Fanuc KAREL source: kb00029.KL

-- PROVISIONAL review KL for V770-1; original PC SHA256 8f31ae490222605812ec860d8ad9381e16546bc304840df08ca040dcb082aeb5
-- Incomplete behavior may be omitted. Consult companion uncertainty JSON. Do not deploy.
PROGRAM KB00029
%NOLOCKGROUP
BEGIN
  -- UNRESOLVED_PC offsets 5-12; opcodes 9D,23
  -- UNRESOLVED_PC offsets 17-26; opcodes 3F,75
  -- UNRESOLVED_PC offsets 31-38; opcodes 9D,23
  -- UNRESOLVED_PC offsets 43-67; opcodes 27,22,22,2A,22,31
  -- UNRESOLVED_PC offsets 72-76; opcodes 7F
END KB00029
